// TIA Portal V20 export
TYPE "UDT_HMI_SeñalesBarreras"
   STRUCT
      MS_11 : Bool;
      MS_12 : Bool;
      MS_21 : Bool;
      MS_22 : Bool;
      STOP : Bool;
      FREE : Bool;
      ENABLE : Bool;
      ACK : Bool;
      Q : Bool;
      MUTING : Bool;
      ACK_REQ : Bool;
      FAULT : Bool;
      Reserva_14 : Bool;
      Reserva_15 : Bool;
      Reserva_16 : Bool;
      Reserva_17 : Bool;
   END_STRUCT;
END_TYPE
